(* PLC project MQTT, Beckhoff Automation GmbH TwinCAT PLC Control 3.5.13.20 *)
(* stored: creationDateTime 2021-01-27T09:57:57.6740367, modificationDateTime 2021-01-27T09:57:57.6740367 *)

PROGRAM PrgMQTTPublish
//Uebergabevariablen an die Funktion beim Aufruf
VAR_INPUT
	sTopicPub : STRING(255);
	mqtt_payload : REAL;
END_VAR

//Variablen innerhalb der Funktion
VAR
	fbMqttClient : FB_IotMqttClient;
	bSetParameter : BOOL := TRUE;
	bConnect : BOOL := TRUE;
	
	(* published message *)
	sPayloadPub : STRING(255);
	fbTimer : TON := (PT:=GVL_MQTT.mqtt_interval);

	hrErrorOccurred : HRESULT; // contains the latest occurred error
END_VAR

            IF bSetParameter THEN
	bSetParameter := FALSE;
	fbMqttClient.sHostName:= GVL_MQTT.mqtt_broker;
	fbMqttClient.nHostPort:= GVL_MQTT.mqtt_port;
	fbMqttClient.sTopicPrefix:= ''; 
	fbMqttClient.sUserName:= GVL_MQTT.username;
	fbMqttClient.sUserPassword:= GVL_MQTT.password;
	
	//Nicht verwendete MQTT Parameter
//	fbMqttClient.nKeepAlive:= 60; 
//	fbMqttClient.sClientId:= 'MyTcMqttClient';  
//	fbMqttClient.stWill:= ; 
//	fbMqttClient.stTLS:= ;
//	fbMqttClient.ipMessageQueue := fbMessageQueue;
END_IF

fbMqttClient.Execute(bConnect);
IF fbMqttClient.bError THEN
	// add your error logging here
	hrErrorOccurred := fbMqttClient.hrErrorCode;
END_IF

IF fbMqttClient.bConnected THEN
	fbTimer(IN:=TRUE);
	IF fbTimer.Q THEN // publish new payload every GVL.mqtt_interval
		fbTimer(IN:=FALSE);
		sPayloadPub := TO_STRING(mqtt_payload);
		fbMqttClient.Publish(	sTopic:= sTopicPub, 
								pPayload:= ADR(sPayloadPub), nPayloadSize:= LEN2(ADR(sPayloadPub))+1, 
								eQoS:= TcIotMqttQos.AtMostOnceDelivery, bRetain:= FALSE, bQueue:= FALSE );
		IF fbMqttClient.bError THEN
			// add your error logging here
			hrErrorOccurred := fbMqttClient.hrErrorCode;
		END_IF
	END_IF
END_IF
          
END_PROGRAM
